// TIA Portal V16 export
// export: Created 2025-05-30T16:35:49.8128107Z, ExportSetting WithDefaults, DisplayName Totally Integrated Automation Portal, DisplayVersion V16, DisplayName TIA Portal Version Control Interface, DisplayVersion V16, DisplayName TIA Portal Openness, DisplayVersion V16, DisplayName STEP 7 Professional, DisplayVersion V16, DisplayName STEP 7 Safety, DisplayVersion V16, DisplayName WinCC Advanced, DisplayVersion V16
FUNCTION "5 - Prog. 3" : Void   // FC3, LAD
TITLE = System Program 3
VERSION : 0.1
// stored: AutoNumber true, IsIECCheckEnabled false, UDAEnableTagReadback false
BEGIN

REGION Network 1: Close 1 Magazine Hole (cilinder)
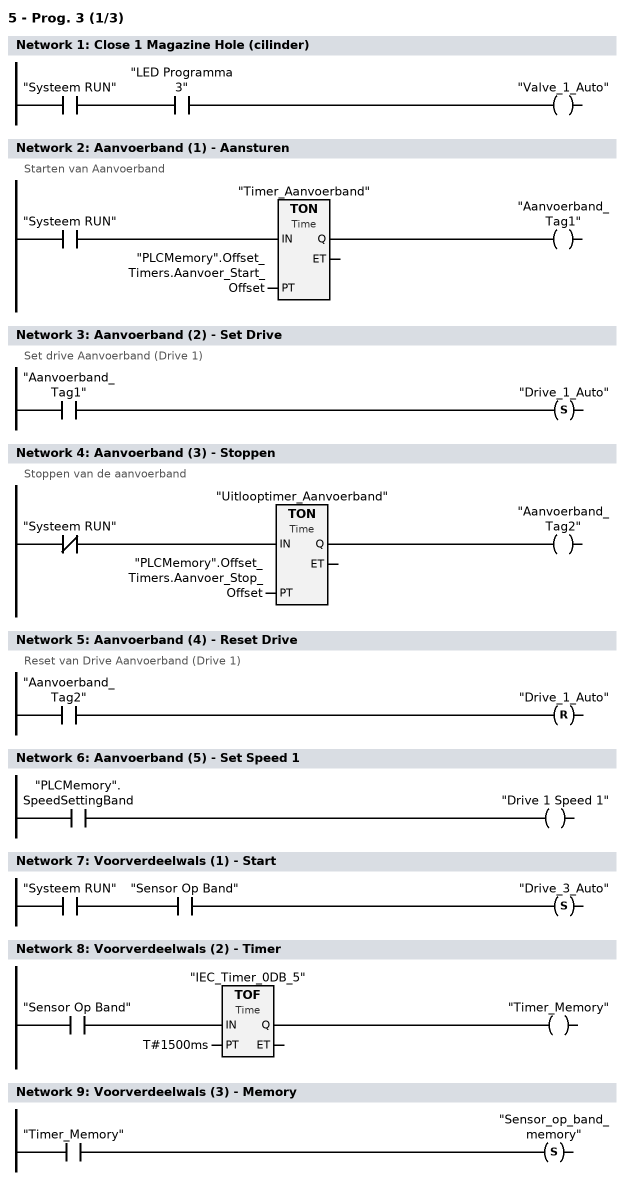
   RUNG wire#powerrail
      Contact( "Systeem RUN" )
      Contact( "LED Programma 3" )
      Coil( "Valve_1_Auto" )
   END_RUNG
   // the same network as SCL:
   "Valve_1_Auto" := "Systeem RUN" AND "LED Programma 3";
END_REGION

REGION Network 2: Aanvoerband (1) - Aansturen
   // Starten van Aanvoerband
   RUNG wire#powerrail
      Contact( "Systeem RUN" )
      { S7_Templates := "time_type := Time" } "Timer_Aanvoerband".TON(pt := "PLCMemory".Offset_Timers.Aanvoer_Start_Offset, et =>)
      Coil( "Aanvoerband_Tag1" )
   END_RUNG
   // the same network as SCL:
   "Timer_Aanvoerband".TON(IN := "Systeem RUN", PT := "PLCMemory".Offset_Timers.Aanvoer_Start_Offset);
   "Aanvoerband_Tag1" := "Timer_Aanvoerband".Q;
END_REGION

REGION Network 3: Aanvoerband (2) - Set Drive
   // Set drive Aanvoerband (Drive 1)
   RUNG wire#powerrail
      Contact( "Aanvoerband_Tag1" )
      S_Coil( "Drive_1_Auto" )
   END_RUNG
   // the same network as SCL:
   IF "Aanvoerband_Tag1" THEN "Drive_1_Auto" := TRUE; END_IF;
END_REGION

REGION Network 4: Aanvoerband (3) - Stoppen
   // Stoppen van de aanvoerband
   RUNG wire#powerrail
      I_Contact( "Systeem RUN" )
      { S7_Templates := "time_type := Time" } "Uitlooptimer_Aanvoerband".TON(pt := "PLCMemory".Offset_Timers.Aanvoer_Stop_Offset, et =>)
      Coil( "Aanvoerband_Tag2" )
   END_RUNG
   // the same network as SCL:
   "Uitlooptimer_Aanvoerband".TON(IN := NOT "Systeem RUN", PT := "PLCMemory".Offset_Timers.Aanvoer_Stop_Offset);
   "Aanvoerband_Tag2" := "Uitlooptimer_Aanvoerband".Q;
END_REGION

REGION Network 5: Aanvoerband (4) - Reset Drive
   // Reset van Drive Aanvoerband (Drive 1)
   RUNG wire#powerrail
      Contact( "Aanvoerband_Tag2" )
      R_Coil( "Drive_1_Auto" )
   END_RUNG
   // the same network as SCL:
   IF "Aanvoerband_Tag2" THEN "Drive_1_Auto" := FALSE; END_IF;
END_REGION

REGION Network 6: Aanvoerband (5) - Set Speed 1
   RUNG wire#powerrail
      Contact( "PLCMemory".SpeedSettingBand )
      Coil( "Drive 1 Speed 1" )
   END_RUNG
   // the same network as SCL:
   "Drive 1 Speed 1" := "PLCMemory".SpeedSettingBand;
END_REGION

REGION Network 7: Voorverdeelwals (1) - Start
   RUNG wire#powerrail
      Contact( "Systeem RUN" )
      Contact( "Sensor Op Band" )
      S_Coil( "Drive_3_Auto" )
   END_RUNG
   // the same network as SCL:
   IF "Systeem RUN" AND "Sensor Op Band" THEN "Drive_3_Auto" := TRUE; END_IF;
END_REGION

REGION Network 8: Voorverdeelwals (2) - Timer
   RUNG wire#powerrail
      Contact( "Sensor Op Band" )
      { S7_Templates := "time_type := Time" } "IEC_Timer_0DB_5".TOF(pt := T#1500ms, et =>)
      Coil( "Timer_Memory" )
   END_RUNG
   // the same network as SCL:
   "IEC_Timer_0DB_5".TOF(IN := "Sensor Op Band", PT := T#1500ms);
   "Timer_Memory" := "IEC_Timer_0DB_5".Q;
END_REGION

REGION Network 9: Voorverdeelwals (3) - Memory
   RUNG wire#powerrail
      Contact( "Timer_Memory" )
      S_Coil( "Sensor_op_band_memory" )
   END_RUNG
   // the same network as SCL:
   IF "Timer_Memory" THEN "Sensor_op_band_memory" := TRUE; END_IF;
END_REGION

REGION Network 10: Voorverdeelwals (4) - Delaying
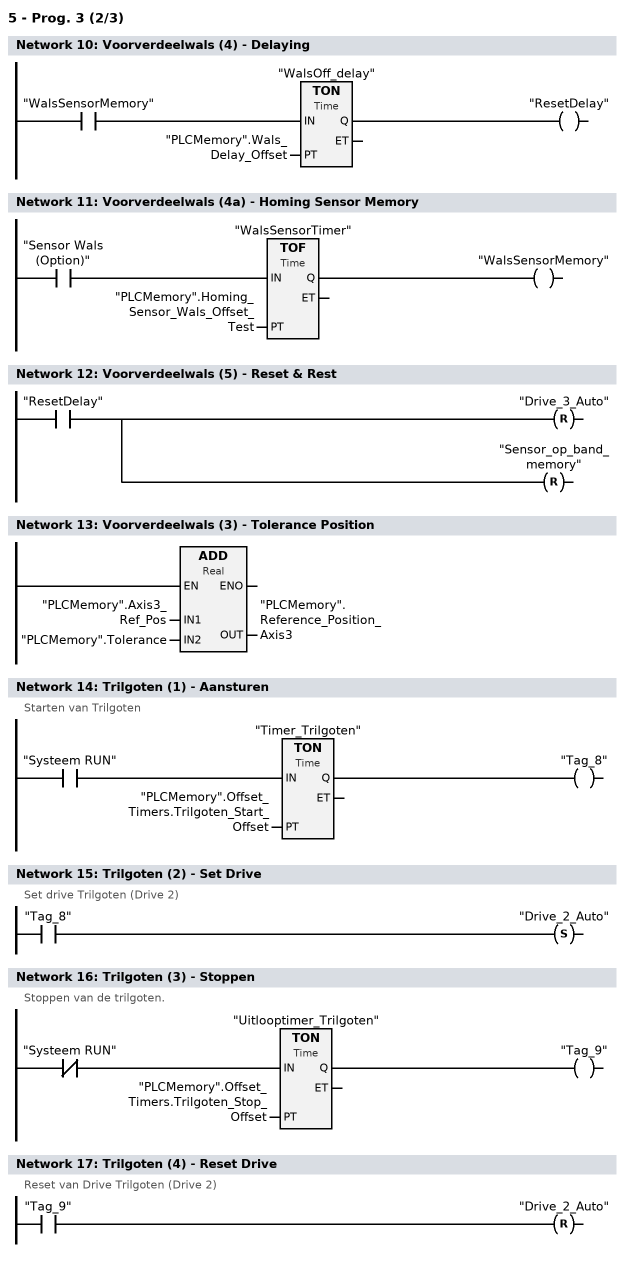
   RUNG wire#powerrail
      Contact( "WalsSensorMemory" )
      { S7_Templates := "time_type := Time" } "WalsOff_delay".TON(pt := "PLCMemory".Wals_Delay_Offset, et =>)
      Coil( "ResetDelay" )
   END_RUNG
   // the same network as SCL:
   "WalsOff_delay".TON(IN := "WalsSensorMemory", PT := "PLCMemory".Wals_Delay_Offset);
   "ResetDelay" := "WalsOff_delay".Q;
END_REGION

REGION Network 11: Voorverdeelwals (4a) - Homing Sensor Memory
   RUNG wire#powerrail
      Contact( "Sensor Wals (Option)" )
      { S7_Templates := "time_type := Time" } "WalsSensorTimer".TOF(pt := "PLCMemory".Homing_Sensor_Wals_Offset_Test, et =>)
      Coil( "WalsSensorMemory" )
   END_RUNG
   // the same network as SCL:
   "WalsSensorTimer".TOF(IN := "Sensor Wals (Option)", PT := "PLCMemory".Homing_Sensor_Wals_Offset_Test);
   "WalsSensorMemory" := "WalsSensorTimer".Q;
END_REGION

REGION Network 12: Voorverdeelwals (5) - Reset & Rest
   RUNG wire#powerrail
      Contact( "ResetDelay" )
      wire#w1
      R_Coil( "Drive_3_Auto" )
   END_RUNG
   RUNG wire#w1
      R_Coil( "Sensor_op_band_memory" )
   END_RUNG
   // the same network as SCL:
   IF "ResetDelay" THEN
       "Drive_3_Auto" := FALSE;
       "Sensor_op_band_memory" := FALSE;
   END_IF;
END_REGION

REGION Network 13: Voorverdeelwals (3) - Tolerance Position
   RUNG wire#powerrail
      { S7_Templates := "SrcType := Real"; S7_GenerateENO := "TRUE" } Add(in1 := "PLCMemory".Axis3_Ref_Pos, in2 := "PLCMemory".Tolerance, out => "PLCMemory".Reference_Position_Axis3)
   END_RUNG
   // the same network as SCL:
   "PLCMemory".Reference_Position_Axis3 := "PLCMemory".Axis3_Ref_Pos + "PLCMemory".Tolerance;
END_REGION

REGION Network 14: Trilgoten (1) - Aansturen
   // Starten van Trilgoten
   RUNG wire#powerrail
      Contact( "Systeem RUN" )
      { S7_Templates := "time_type := Time" } "Timer_Trilgoten".TON(pt := "PLCMemory".Offset_Timers.Trilgoten_Start_Offset, et =>)
      Coil( "Tag_8" )
   END_RUNG
   // the same network as SCL:
   "Timer_Trilgoten".TON(IN := "Systeem RUN", PT := "PLCMemory".Offset_Timers.Trilgoten_Start_Offset);
   "Tag_8" := "Timer_Trilgoten".Q;
END_REGION

REGION Network 15: Trilgoten (2) - Set Drive
   // Set drive Trilgoten (Drive 2)
   RUNG wire#powerrail
      Contact( "Tag_8" )
      S_Coil( "Drive_2_Auto" )
   END_RUNG
   // the same network as SCL:
   IF "Tag_8" THEN "Drive_2_Auto" := TRUE; END_IF;
END_REGION

REGION Network 16: Trilgoten (3) - Stoppen
   // Stoppen van de trilgoten.
   RUNG wire#powerrail
      I_Contact( "Systeem RUN" )
      { S7_Templates := "time_type := Time" } "Uitlooptimer_Trilgoten".TON(pt := "PLCMemory".Offset_Timers.Trilgoten_Stop_Offset, et =>)
      Coil( "Tag_9" )
   END_RUNG
   // the same network as SCL:
   "Uitlooptimer_Trilgoten".TON(IN := NOT "Systeem RUN", PT := "PLCMemory".Offset_Timers.Trilgoten_Stop_Offset);
   "Tag_9" := "Uitlooptimer_Trilgoten".Q;
END_REGION

REGION Network 17: Trilgoten (4) - Reset Drive
   // Reset van Drive Trilgoten (Drive 2)
   RUNG wire#powerrail
      Contact( "Tag_9" )
      R_Coil( "Drive_2_Auto" )
   END_RUNG
   // the same network as SCL:
   IF "Tag_9" THEN "Drive_2_Auto" := FALSE; END_IF;
END_REGION

REGION Network 18: Overname (1) - Set Timing as Drive 1
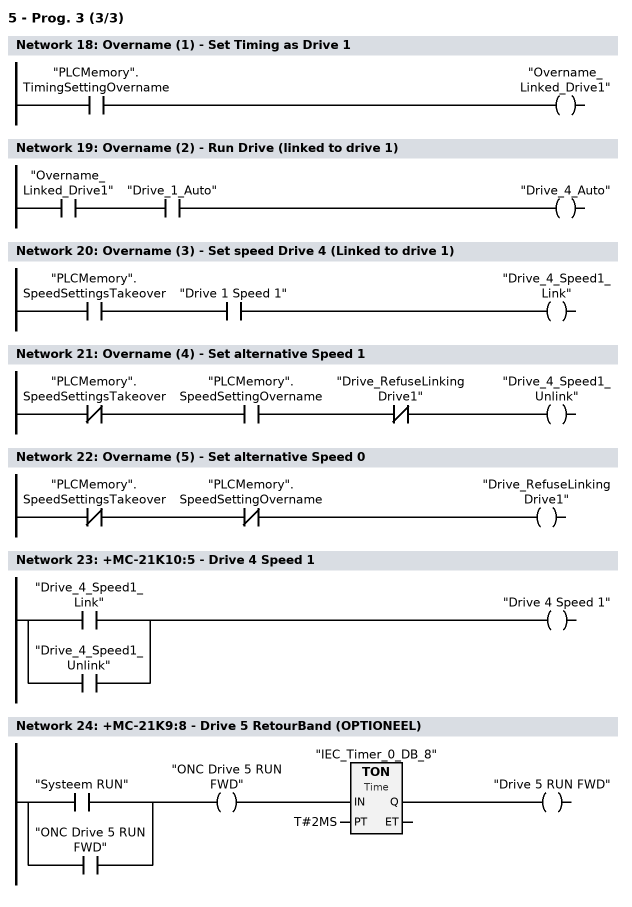
   RUNG wire#powerrail
      Contact( "PLCMemory".TimingSettingOvername )
      Coil( "Overname_Linked_Drive1" )
   END_RUNG
   // the same network as SCL:
   "Overname_Linked_Drive1" := "PLCMemory".TimingSettingOvername;
END_REGION

REGION Network 19: Overname (2) - Run Drive (linked to drive 1)
   RUNG wire#powerrail
      Contact( "Overname_Linked_Drive1" )
      Contact( "Drive_1_Auto" )
      Coil( "Drive_4_Auto" )
   END_RUNG
   // the same network as SCL:
   "Drive_4_Auto" := "Overname_Linked_Drive1" AND "Drive_1_Auto";
END_REGION

REGION Network 20: Overname (3) - Set speed Drive 4 (Linked to drive 1)
   RUNG wire#powerrail
      Contact( "PLCMemory".SpeedSettingsTakeover )
      Contact( "Drive 1 Speed 1" )
      Coil( "Drive_4_Speed1_Link" )
   END_RUNG
   // the same network as SCL:
   "Drive_4_Speed1_Link" := "PLCMemory".SpeedSettingsTakeover AND "Drive 1 Speed 1";
END_REGION

REGION Network 21: Overname (4) - Set alternative Speed 1
   RUNG wire#powerrail
      I_Contact( "PLCMemory".SpeedSettingsTakeover )
      Contact( "PLCMemory".SpeedSettingOvername )
      I_Contact( "Drive_RefuseLinkingDrive1" )
      Coil( "Drive_4_Speed1_Unlink" )
   END_RUNG
   // the same network as SCL:
   "Drive_4_Speed1_Unlink" := NOT "PLCMemory".SpeedSettingsTakeover AND "PLCMemory".SpeedSettingOvername AND NOT "Drive_RefuseLinkingDrive1";
END_REGION

REGION Network 22: Overname (5) - Set alternative Speed 0
   RUNG wire#powerrail
      I_Contact( "PLCMemory".SpeedSettingsTakeover )
      I_Contact( "PLCMemory".SpeedSettingOvername )
      Coil( "Drive_RefuseLinkingDrive1" )
   END_RUNG
   // the same network as SCL:
   "Drive_RefuseLinkingDrive1" := NOT "PLCMemory".SpeedSettingsTakeover AND NOT "PLCMemory".SpeedSettingOvername;
END_REGION

REGION Network 23: +MC-21K10:5 - Drive 4 Speed 1
   RUNG wire#powerrail
      Contact( "Drive_4_Speed1_Link" )
      wire#w1
      Coil( "Drive 4 Speed 1" )
   END_RUNG
   RUNG wire#powerrail
      Contact( "Drive_4_Speed1_Unlink" )
   END_RUNG wire#w1
   // the same network as SCL:
   "Drive 4 Speed 1" := "Drive_4_Speed1_Link" OR "Drive_4_Speed1_Unlink";
END_REGION

REGION Network 24: +MC-21K9:8 - Drive 5 RetourBand (OPTIONEEL)
   RUNG wire#powerrail
      Contact( "Systeem RUN" )
      wire#w1
      Coil( "ONC Drive 5 RUN FWD" )
      { S7_Templates := "time_type := Time" } "IEC_Timer_0_DB_8".TON(pt := T#2MS, et =>)
      Coil( "Drive 5 RUN FWD" )
   END_RUNG
   RUNG wire#powerrail
      Contact( "ONC Drive 5 RUN FWD" )
   END_RUNG wire#w1
   // the same network as SCL:
   "ONC Drive 5 RUN FWD" := "Systeem RUN" OR "ONC Drive 5 RUN FWD";
   "IEC_Timer_0_DB_8".TON(IN := "ONC Drive 5 RUN FWD", PT := T#2MS);
   "Drive 5 RUN FWD" := "IEC_Timer_0_DB_8".Q;
END_REGION
END_FUNCTION
